{attribute addProperty BoxType "AX8620-0000-0027"}
{attribute addProperty Id "StatuswordAT %I*Statusword_177FE35F162"}
{attribute addProperty CRC "3243559737"}
{attribute addProperty SizeInBites "16"}
{attribute addProperty SizeInBytes "2"}
TYPE PSM_Statusword_C154CB39 :
STRUCT
	{attribute addProperty Name "Statusword"}
	Statusword AT %I* : Statusword_177FE35F;
END_STRUCT
END_TYPE

(* stored: Version 1.2.0.0, ProductVersion 3.1.4024.9
   DUT PSM_Statusword_C154CB39: Id {fa99e4fc-891a-4e0f-8daa-b22cd289912a} *)
